{attribute 'GeneratedUsingTerminal: EL5101-0000-1020'}
{attribute addProperty BoxType "EL5101-0000-1020"}
{attribute addProperty Id "Enable_latch_CBOOL1Enable_latch_extern_on_positive_edgeBOOL1Set_counterBOOL1Enable_latch_extern_on_negative_edgeBOOL1"}
{attribute addProperty CRC "1861404112"}
{attribute addProperty Size "4"}
TYPE Control_6EF2C5D0 :
STRUCT
	{attribute addProperty Name "Enable_latch_C"}
	Enable_latch_C : BOOL;
	{attribute addProperty Name "Enable_latch_extern_on_positive_edge"}
	Enable_latch_extern_on_positive_edge : BOOL;
	{attribute addProperty Name "Set_counter"}
	Set_counter : BOOL;
	{attribute addProperty Name "Enable_latch_extern_on_negative_edge"}
	Enable_latch_extern_on_negative_edge : BOOL;
END_STRUCT
END_TYPE

(* stored: Version 1.2.0.0, ProductVersion 3.1.4024.9
   DUT Control_6EF2C5D0: Id {5141b583-aca6-49f6-98cb-6d3989fbbbc1} *)
